SYSTEM washer_detector
  (* Version 1.0, 2024-11-25, obotnar *)
  APPLICATION washer_detectorApp
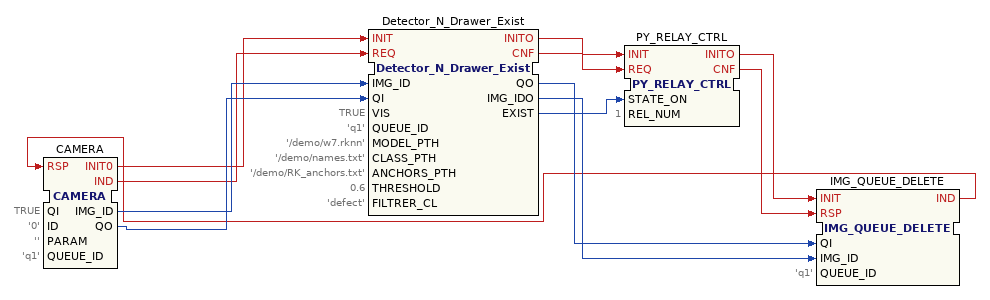
    FBS
      CAMERA : CAMERA(QI := TRUE, ID := '0', PARAM := '', QUEUE_ID := 'q1');
      IMG_QUEUE_DELETE : IMG_QUEUE_DELETE(QUEUE_ID := 'q1');
      Detector_N_Drawer_Exist : Detector_N_Drawer_Exist(VIS := TRUE, QUEUE_ID := 'q1', MODEL_PTH := '/demo/w7.rknn', CLASS_PTH := '/demo/names.txt', ANCHORS_PTH := '/demo/RK_anchors.txt', THRESHOLD := 0.6, FILTRER_CL := 'defect');
      PY_RELAY_CTRL : PY_RELAY_CTRL(REL_NUM := 1);
    END_FBS
    EVENT_CONNECTIONS
      CAMERA.INIT0 TO Detector_N_Drawer_Exist.INIT;
      CAMERA.IND TO Detector_N_Drawer_Exist.REQ;
      IMG_QUEUE_DELETE.IND TO CAMERA.RSP;
      Detector_N_Drawer_Exist.INITO TO PY_RELAY_CTRL.INIT;
      Detector_N_Drawer_Exist.CNF TO PY_RELAY_CTRL.REQ;
      PY_RELAY_CTRL.INITO TO IMG_QUEUE_DELETE.INIT;
      PY_RELAY_CTRL.CNF TO IMG_QUEUE_DELETE.RSP;
    END_CONNECTIONS
    DATA_CONNECTIONS
      CAMERA.IMG_ID TO Detector_N_Drawer_Exist.IMG_ID;
      CAMERA.QO TO Detector_N_Drawer_Exist.QI;
      Detector_N_Drawer_Exist.QO TO IMG_QUEUE_DELETE.QI;
      Detector_N_Drawer_Exist.IMG_IDO TO IMG_QUEUE_DELETE.IMG_ID;
      Detector_N_Drawer_Exist.EXIST TO PY_RELAY_CTRL.STATE_ON;
    END_CONNECTIONS
  END_APPLICATION
  DEVICE FORTE_PC : FORTE_PC(MGR_ID := "10.5.20.198:62499" (* Device manager socket ID *))
    {SET_ATTRIBUTE(Profile, HOLOBLOC)}
    RESOURCE EMB_RES : EMB_RES
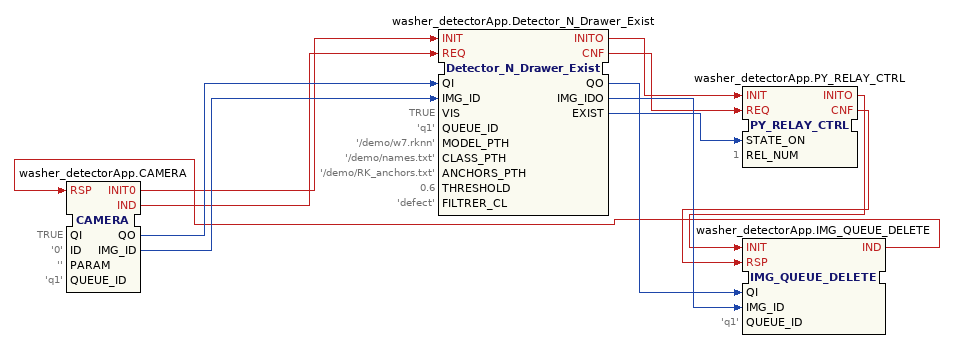
      FBS
        washer_detectorApp.CAMERA : CAMERA(QI := TRUE, ID := '0', PARAM := '', QUEUE_ID := 'q1');
        washer_detectorApp.IMG_QUEUE_DELETE : IMG_QUEUE_DELETE(QUEUE_ID := 'q1');
        washer_detectorApp.Detector_N_Drawer_Exist : Detector_N_Drawer_Exist(VIS := TRUE, QUEUE_ID := 'q1', MODEL_PTH := '/demo/w7.rknn', CLASS_PTH := '/demo/names.txt', ANCHORS_PTH := '/demo/RK_anchors.txt', THRESHOLD := 0.6, FILTRER_CL := 'defect');
        washer_detectorApp.PY_RELAY_CTRL : PY_RELAY_CTRL(REL_NUM := 1);
      END_FBS
      EVENT_CONNECTIONS
        washer_detectorApp.CAMERA.INIT0 TO washer_detectorApp.Detector_N_Drawer_Exist.INIT;
        washer_detectorApp.CAMERA.IND TO washer_detectorApp.Detector_N_Drawer_Exist.REQ;
        washer_detectorApp.IMG_QUEUE_DELETE.IND TO washer_detectorApp.CAMERA.RSP;
        washer_detectorApp.Detector_N_Drawer_Exist.INITO TO washer_detectorApp.PY_RELAY_CTRL.INIT;
        washer_detectorApp.Detector_N_Drawer_Exist.CNF TO washer_detectorApp.PY_RELAY_CTRL.REQ;
        washer_detectorApp.PY_RELAY_CTRL.INITO TO washer_detectorApp.IMG_QUEUE_DELETE.INIT;
        washer_detectorApp.PY_RELAY_CTRL.CNF TO washer_detectorApp.IMG_QUEUE_DELETE.RSP;
      END_CONNECTIONS
      DATA_CONNECTIONS
        washer_detectorApp.CAMERA.QO TO washer_detectorApp.Detector_N_Drawer_Exist.QI;
        washer_detectorApp.CAMERA.IMG_ID TO washer_detectorApp.Detector_N_Drawer_Exist.IMG_ID;
        washer_detectorApp.Detector_N_Drawer_Exist.QO TO washer_detectorApp.IMG_QUEUE_DELETE.QI;
        washer_detectorApp.Detector_N_Drawer_Exist.IMG_IDO TO washer_detectorApp.IMG_QUEUE_DELETE.IMG_ID;
        washer_detectorApp.Detector_N_Drawer_Exist.EXIST TO washer_detectorApp.PY_RELAY_CTRL.STATE_ON;
      END_CONNECTIONS
    END_RESOURCE
  END_DEVICE
  MAPPINGS
    washer_detectorApp.CAMERA ON FORTE_PC.EMB_RES;
    washer_detectorApp.IMG_QUEUE_DELETE ON FORTE_PC.EMB_RES;
    washer_detectorApp.Detector_N_Drawer_Exist ON FORTE_PC.EMB_RES;
    washer_detectorApp.PY_RELAY_CTRL ON FORTE_PC.EMB_RES;
  END_MAPPINGS
  SEGMENTS
    Ethernet : Ethernet;
  END_SEGMENTS
  LINKS
    FORTE_PC => Ethernet;
  END_LINKS
END_SYSTEM
